KUKA KRL program: rechazo_bal.src, rechazo_bal.dat

--- rechazo_bal.src ---
&ACCESS RVO4
&REL 20
&PARAM TEMPLATE = C:\KRC\Roboter\Template\vorgabe
&PARAM EDITMASK = *
DEF rechazo_bal( )

;================================================
; MODELO   : C-520
; IE GRUPO : 5J
; ESTACION : 85
; ROBOT    : 85r01
; FUNCION  : xxxxxxx
;================================================

;FOLD INI
  ;FOLD BASISTECH INI
    GLOBAL INTERRUPT DECL 3 WHEN $STOPMESS==TRUE DO IR_STOPM ( )
    INTERRUPT ON 3
    BAS (#INITMOV,0 )
  ;ENDFOLD (BASISTECH INI)
;FOLD SPOTTECH INI
;USERSPOT(#INIT)
;ENDFOLD (SPOTTECH INI)
;FOLD GRIPPERTECH INI
USER_GRP(0,DUMMY,DUMMY,GDEFAULT)
INTERRUPT DECL 20 WHEN $FLAG[20]==FALSE DO GRPS(#MON_ERR,20)
;ENDFOLD (GRIPPERTECH INI)
  ;FOLD USER INI
    ;Make your modifications here

  ;ENDFOLD (USER INI)
;ENDFOLD (INI)

;FOLD OUT 34 'PETICION A DISPOSITIVO 2' State=FALSE ;%{PE}%R 5.6.13,%MKUKATPBASIS,%COUT,%VOUTX,%P 2:34, 3:PETICION A DISPOSITIVO 2, 5:FALSE, 6:
$OUT[34]=FALSE
;ENDFOLD
;FOLD OUT 35 'PETICION A DISPOSITIVO 3' State=FALSE ;%{PE}%R 5.6.13,%MKUKATPBASIS,%COUT,%VOUTX,%P 2:35, 3:PETICION A DISPOSITIVO 3, 5:FALSE, 6:
$OUT[35]=FALSE
;ENDFOLD

;FOLD OUT 38 'PETICION A DISPOSITIVO 6' State=FALSE ;%{PE}%R 5.6.13,%MKUKATPBASIS,%COUT,%VOUTX,%P 2:38, 3:PETICION A DISPOSITIVO 6, 5:FALSE, 6:
$OUT[38]=FALSE
;ENDFOLD
;punto retirada
;FOLD PTP P1 Vel=100 % PDAT1 Tool[14]:camara Base[0];%{PE}%R 5.6.13,%MKUKATPBASIS,%CMOVE,%VPTP,%P 1:PTP, 2:P1, 3:, 5:100, 7:PDAT1
$BWDSTART=FALSE
PDAT_ACT=PPDAT1
FDAT_ACT=FP1
BAS(#PTP_PARAMS,100)
PTP XP1
;ENDFOLD

;FOLD OUT 19 'LIBERACION AREA 3 ems inf' State=TRUE ;%{PE}%R 5.6.13,%MKUKATPBASIS,%COUT,%VOUTX,%P 2:19, 3:LIBERACION AREA 3 ems inf, 5:TRUE, 6:
$OUT[19]=TRUE
;ENDFOLD
;FOLD OUT 18 'LIBERACION AREA 2 ems sup' State=TRUE ;%{PE}%R 5.6.13,%MKUKATPBASIS,%COUT,%VOUTX,%P 2:18, 3:LIBERACION AREA 2 ems sup, 5:TRUE, 6:
$OUT[18]=TRUE
;ENDFOLD
;FOLD OUT 42 'TRABAJO FINALIZADO 2' State=FALSE ;%{PE}%R 5.6.13,%MKUKATPBASIS,%COUT,%VOUTX,%P 2:42, 3:TRABAJO FINALIZADO 2, 5:FALSE, 6:
$OUT[42]=FALSE
;ENDFOLD

;FOLD OUT 40 'PETICION A DISPOSITIVO 8' State=TRUE ;%{PE}%R 5.6.13,%MKUKATPBASIS,%COUT,%VOUTX,%P 2:40, 3:PETICION A DISPOSITIVO 8, 5:TRUE, 6:
$OUT[40]=TRUE
;ENDFOLD
;FOLD WAIT FOR ( IN 40 'PERMISO DISPOSITIVO 8' );%{PE}%R 5.6.13,%MKUKATPBASIS,%CEXT_WAIT_FOR,%VEXT_WAIT_FOR,%P 2:, 4:, 5:$IN, 6:40, 7:PERMISO DISPOSITIVO 8, 9:
WAIT FOR  ( $IN[40] )
;ENDFOLD
;FOLD OUT 40 'PETICION A DISPOSITIVO 8' State=FALSE ;%{PE}%R 5.6.13,%MKUKATPBASIS,%COUT,%VOUTX,%P 2:40, 3:PETICION A DISPOSITIVO 8, 5:FALSE, 6:
$OUT[40]=FALSE
;ENDFOLD

SALTO_RECHAZO=TRUE
END

--- rechazo_bal.dat ---
&ACCESS RVO4
&REL 20
&PARAM TEMPLATE = C:\KRC\Roboter\Template\vorgabe
&PARAM EDITMASK = *
DEFDAT  RECHAZO_BAL
;FOLD EXTERNAL DECLARATIONS;%{PE}%MKUKATPBASIS,%CEXT,%VCOMMON,%P
;FOLD GRIPPERTECH EXT
EXT  H50 (INT  :IN,INT  :IN,INT  :IN,GRP_TYP  :IN )
;ENDFOLD (GRIPPERTECH EXT)
;FOLD SPOTTECH EXT
EXT  USERSPOT (S_COMMAND  :IN,SPOT_TYPE  :IN )
;ENDFOLD (SPOTTECH EXT)
;FOLD BASISTECH EXT;%{PE}%MKUKATPBASIS,%CEXT,%VEXT,%P
EXT  BAS (BAS_COMMAND  :IN,REAL  :IN )
DECL INT SUCCESS
;ENDFOLD (BASISTECH EXT)
;FOLD USER EXT;%{E}%MKUKATPUSER,%CEXT,%VEXT,%P
;Make here your modifications

;ENDFOLD (USER EXT)
;ENDFOLD (EXTERNAL DECLARATIONS)
DECL BASIS_SUGG_T LAST_BASIS={POINT1[] "P1                      ",POINT2[] "P1                      ",CP_PARAMS[] "CPDAT0                  ",PTP_PARAMS[] "PDAT1                   ",CONT[] "                        ",CP_VEL[] "2.0                     ",PTP_VEL[] "100                     ",SYNC_PARAMS[] "SYNCDAT                 ",SPL_NAME[] "S0                      "}
DECL E6POS XP1={X 450.707703,Y 1172.57898,Z 1337.21399,A -97.1499176,B 88.7769928,C 102.053902,S 2,T 11,E1 0.0,E2 0.0,E3 0.0,E4 0.0,E5 0.0,E6 0.0}
DECL FDAT FP1={TOOL_NO 14,BASE_NO 0,IPO_FRAME #BASE,POINT2[] " ",TQ_STATE FALSE}
DECL PDAT PPDAT1={VEL 100.0,ACC 100.0,APO_DIST 100.0}
ENDDAT
